PROGRAM MAIN
VAR
	fbTestBase : FB_TestBase;
	fbTestEquipmentBase	: FB_TestEquipmentBase;
	fbTestEquipmentBase2	: FB_TestEquipmentBase;
	
	AnotherTestAlarmList	: ARRAY[E_TestEquipmentAlarmList.VerboseAlarm..E_TestEquipmentAlarmList.CriticalAlarm] OF ST_EquipmentAlarm;
	
	Reset	: BOOL;
	
	fbSupervistorBase : FB_SupervisorBase;
	
END_VAR

VAR PERSISTENT
	TestManualControl	: ARRAY[1..3] OF BOOL;
	TestName			: ARRAY[1..3] OF STRING(40);
	TestStation			: ARRAY[1..3] OF STRING(40);	
	

END_VAR

fbTestBase.Definition.Name := TestName[1];
fbTestBase.Definition.Station := TestStation[1];
fbTestBase.EnableManualControl := TestManualControl[1];

fbTestBase();

fbTestEquipmentBase.Definition.Name := TestName[2];
fbTestEquipmentBase.Definition.Station := TestStation[2];
fbTestEquipmentBase.EnableManualControl := TestManualControl[2];

fbTestEquipmentBase();

fbTestEquipmentBase2.Definition.Name := TestName[3];
fbTestEquipmentBase2.Definition.Station := TestStation[3];
fbTestEquipmentBase2.EnableManualControl := TestManualControl[3];

fbTestEquipmentBase2();

IF Reset THEN
	fbTestEquipmentBase.Reset();	
	fbTestEquipmentBase2.Reset();
	Reset := FALSE;
END_IF

fbSupervistorBase();

fbSupervistorBase.CompileAlarmList(AlarmListDetails := fbTestEquipmentBase.AlarmListDetails);
fbSupervistorBase.CompileAlarmList(AlarmListDetails := fbTestEquipmentBase2.AlarmListDetails);

END_PROGRAM

(* stored: Version 1.1.0.1
   POU MAIN: Id {72253cc2-044e-4b72-9460-526041b96d44}, SpecialFunc None *)
